(* IEC 61131-3 sources: plc_generation_empirical_study/datasets/packages/internal_v0_1_precalibration_20260810/qualification_only/C07_E01_linear_scaling/negative_control, 1 file *)

(* ---- NC1.st ---- *)
FUNCTION_BLOCK C08_E01_linear_scaling
VAR_INPUT
    Raw : INT;
END_VAR
VAR_OUTPUT
    Engineering : REAL;
END_VAR

Engineering := INT_TO_REAL(Raw) * 0.1;

END_FUNCTION_BLOCK
